// TIA Portal V20 export
VAR_GLOBAL   // PLC tag table "UPS"
   M_ShutdownPCRequest AT %MW2 : Int;
   M_ShutdownPCResponse AT %MW4 : Int;
END_VAR
